// Mitsubishi GX Works2 project: hmi-multi-program_cylinder   PLC: Q02/Q02H

PROGRAM MAIN
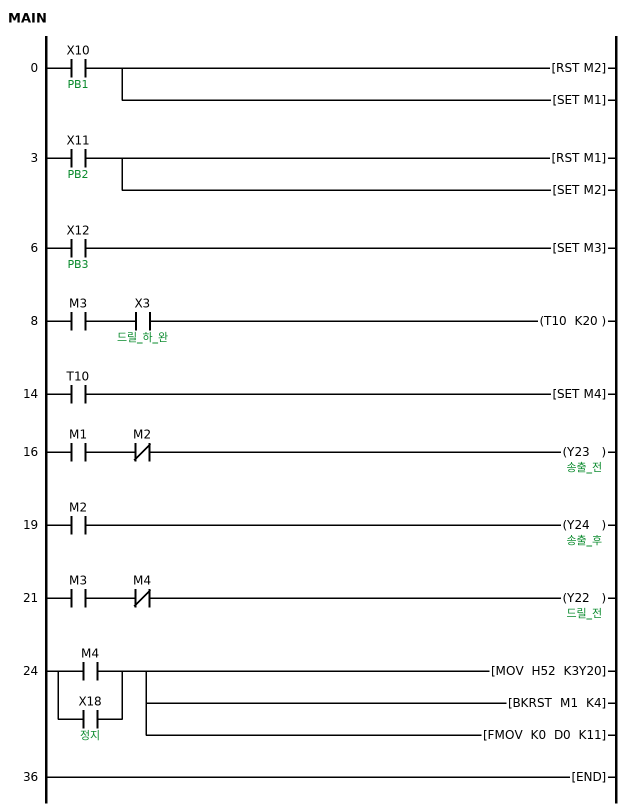
0     LD      X10  ; PB1
      RST     M2
      SET     M1
3     LD      X11  ; PB2
      RST     M1
      SET     M2
6     LD      X12  ; PB3
      SET     M3
8     LD      M3
      AND     X3  ; 드릴_하_완
      OUT     T10 K20
14    LD      T10
      SET     M4
16    LD      M1
      ANI     M2
      OUT     Y23  ; 송출_전
19    LD      M2
      OUT     Y24  ; 송출_후
21    LD      M3
      ANI     M4
      OUT     Y22  ; 드릴_전
24    LD      M4
      OR      X18  ; 정지
      MOV     H52 K3Y20  ; 공급_전
      BKRST   M1 K4
      FMOV    K0 D0 K11
36    END
END_PROGRAM

PROGRAM HMI
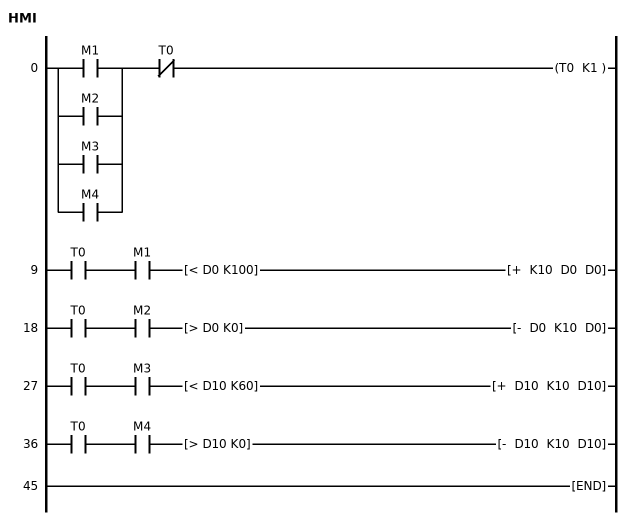
0     LD      M1
      OR      M2
      OR      M3
      OR      M4
      ANI     T0
      OUT     T0 K1
9     LD      T0
      AND     M1
      AND<    D0 K100
      +       K10 D0 D0
18    LD      T0
      AND     M2
      AND>    D0 K0
      -       D0 K10 D0
27    LD      T0
      AND     M3
      AND<    D10 K60
      +       D10 K10 D10
36    LD      T0
      AND     M4
      AND>    D10 K0
      -       D10 K10 D10
45    END
END_PROGRAM

PROGRAM ALARM
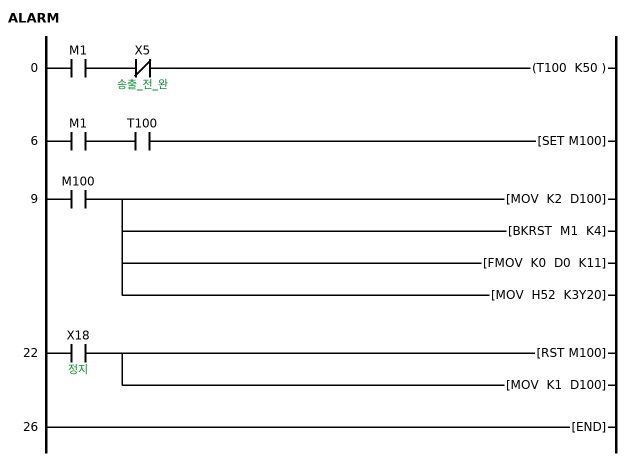
0     LD      M1
      ANI     X5  ; 송출_전_완
      OUT     T100 K50
6     LD      M1
      AND     T100
      SET     M100
9     LD      M100
      MOV     K2 D100
      BKRST   M1 K4
      FMOV    K0 D0 K11
      MOV     H52 K3Y20  ; 공급_전
22    LD      X18  ; 정지
      RST     M100
      MOV     K1 D100
26    END
END_PROGRAM

// device comments not shown above
X0  ; 공급_후_완
X1  ; 공급_전_완
X2  ; 드릴_상_완
X4  ; 송출_후_완
X6  ; 배출_후_완
X7  ; 배출_전_완
X8  ; 매거진
X9  ; 비금속
X0A  ; 금속
Y21  ; 공급_후
Y25  ; 배출_전
Y26  ; 배출_후
Y27  ; 컨베이어
Y28  ; 가공도
Y29  ; 적색
Y2A  ; 황색
Y2B  ; 녹색
